// Count all event class related objects with active events.
FUNCTION F_ObserveEventClass  :UINT
VAR_INPUT
	nEventClassID		: UINT					:= 0;		// Target event class ID.
END_VAR
VAR
	_nEvents			:	UINT;
	_iObj				: I_BA_Object;
	_iEvtObj			: I_BA_EventObject;
END_VAR

// Iterate over all objects:
_nEvents := 0;
WHILE (F_BA_IterateObjects(_iObj)) DO
	IF (NOT __QUERYINTERFACE(_iObj,_iEvtObj)) THEN
		;	     
	ELSIF (_iEvtObj.EventClassID <> nEventClassID) THEN
		; // Skip.
	ELSIF (_iEvtObj.Event = FALSE) THEN
		; // Skip.
	ELSE
		_nEvents := _nEvents+1;
	END_IF
END_WHILE
F_ObserveEventClass:=_nEvents;

END_FUNCTION

(* stored: Version 1.1.0.1, ProductVersion 3.1.4026.17
   POU F_ObserveEventClass: Id {370192c2-da90-42d9-8244-fe02d9f057f8}, SpecialFunc None *)
